# EPICS substitutions: db/ecmcEL7037_PosIF.substitutions
file ecmcEcSlave.template
{
  pattern {}
          {}
}

file ecmcEL7037_PosIF.template
{
  pattern {LINR,    ESLO,   EOFF,   EGU,        PREC, LOW, LOLO, HIGH, HIHI, HYST, LLSV,       LSV,        HSV,        HHSV      }
          {"SLOPE", 1,      0,      "Raw",      0,    0,   0,    0,    0,    0,    "NO_ALARM", "NO_ALARM", "NO_ALARM", "NO_ALARM"}
}
